# EPICS autosave request: iocBoot/ioc13ida_pg3/auto_settings.req
file "spinnaker_settings.req",            P=$(P),  R=cam1:
file "NDStdArrays_settings.req",          P=$(P),  R=image1:
file "commonPlugin_settings.req",         P=$(P)
$(P)cam1:GC_OnBoaColProEna
$(P)cam1:GC_VideoMode
$(P)cam1:GC_DevLinThrLimit
$(P)cam1:GC_AcqFrameRateAuto
